// TwinCAT 3 PLC project FMS_201_Monol_tico
// ProgramVersion: 3.1.4024.0
// libraries:
//   Tc2_Standard, * (Beckhoff Automation GmbH)
//   Tc2_System, * (Beckhoff Automation GmbH)
//   Tc3_Module, * (Beckhoff Automation GmbH)
// project tree:
//   / PlcTask.TcTTO
//   POUs/ FB_Clock.TcPOU, FB_Estacion.TcPOU, MAIN.TcPOU (not stored)
// (motion and I/O tree: see PLC project fms_201_manual)
// real-time tasks:
//   TASK PlcTask: cycle T#10ms, priority 20, ADS port 350
//   TASK PlcTask1: cycle T#10ms, priority 21, ADS port 351
//   TASK PlcTask2: cycle T#10ms, priority 22, ADS port 352
//   TASK PlcTask3: cycle T#10ms, priority 23, ADS port 353
//   TASK PlcTask4: cycle T#10ms, priority 24, ADS port 354
//   TASK PlcTask5: cycle T#10ms, priority 25, ADS port 355
//   TASK PlcTask6: cycle T#10ms, priority 26, ADS port 356
// variable links:

CONFIGURATION FMS_201_Monol_tico
    RESOURCE PLC ON TwinCAT3
        TASK PlcTask(INTERVAL := T#10ms, PRIORITY := 23);
        PROGRAM MAIN WITH PlcTask : MAIN;
    END_RESOURCE
END_CONFIGURATION

// ---- POUs/FB_Clock.TcPOU
FUNCTION_BLOCK FB_Clock

VAR_INPUT
	EN: BOOL :=TRUE; 		// Entrada de nuestro temporizador
	PT: TIME := T#500MS;	// Tiempo de nuestro temporizador
END_VAR

VAR_OUTPUT
	ET: TIME;	// Sirve para consultar el tiempo que lleva la entrada PT
	Q: BOOL;	// Salida de nuestro temporizador
END_VAR
VAR
	Timer: TON;
END_VAR

// Función de salida

IF Timer.Q THEN
	Q := NOT Q;
END_IF

// Bloque de función TON
// Definimos la condición de entrada IN cuando EN esté TRUE (siempre) y no esté activa la salida del temporizador
Timer(IN:= EN AND NOT Timer.Q, PT := PT, ET => ET);

END_FUNCTION_BLOCK

// ---- POUs/FB_Estacion.TcPOU
FUNCTION_BLOCK FB_Estacion
VAR_INPUT
	// Parámetros
	TpoEstabilidad: TIME := T#2000MS;
	UdsSolicitadas:UINT := 5;
	
END_VAR
VAR_OUTPUT
	// Parámetros
	CondicionInicial: BOOL;
	UdsPendientes: UINT;
	UdsRealizadas: UINT;
	
	// Entradas comunes
	PulsadorEmergencia AT %I*: BOOL;
    SelectorManual AT %I*: BOOL;
    PulsadorMarcha AT %I*: BOOL;
    PulsadorParada AT %I*: BOOL := TRUE; // Contacto normalmente cerrado
    EstacionConectada AT %I*: BOOL := TRUE;
    DetectorPresion AT %I*: BOOL := TRUE;
	
	PalePresencia AT %I*: BOOL;
    PaleCodigoBit0 AT %I*: BOOL;
    PaleCodigoBit1 AT %I*: BOOL;
    PaleCodigoBit2 AT %I*: BOOL;
	
	// Entradas específicas
	DescargadorDetras AT %I*: BOOL;
	DescargadorDelante AT %I*: BOOL;
	VerticalArriba AT %I*: BOOL;
	VerticalAbajo AT %I*: BOOL;
	VerificadorArriba AT %I*: BOOL;
	VerificadorAbajo AT %I*: BOOL;
	DesplazadorDetras AT %I*: BOOL;
	AlimentadorDetras AT %I*: BOOL;
	AlimentadorDelante AT %I*: BOOL;
	VacioDescargador AT %I*: BOOL;
	PresenciaBaseAlimentador AT %I*:BOOL;
END_VAR
VAR
	// Bloques funcionales
	CLK: FB_Clock;
	// Salidas comunes
	DesconectaEstacion AT %Q*: BOOL;
    LamparaAlarma AT %Q*: BOOL;
    LamparaMarcha AT %Q*: BOOL;
	LamparaFaltaMaterial AT %Q*: BOOL;
    AvisadorSonoro AT %Q*: BOOL;

    CintaMotorActiva AT %Q*: BOOL;
    CintaMotorInvierte AT %Q*: BOOL;
    CintaRetenedorBaja AT %Q*: BOOL;
    CintaSeparadorSube AT %Q*: BOOL;
	
	// Salidas específicas
	DescargadorAtras AT %Q*: BOOL;
	DescargadorAdelante AT %Q*: BOOL;
	DescargadorBaja AT %Q*: BOOL;
	RechazadorAdelante AT %Q*: BOOL;
	VerificadorBaja AT %Q*: BOOL;
	DesplazadorAdelante AT %Q*: BOOL;
	AlimentadorAdelante AT %Q*: BOOL;
	EyectorSucciona AT %Q*: BOOL;
END_VAR

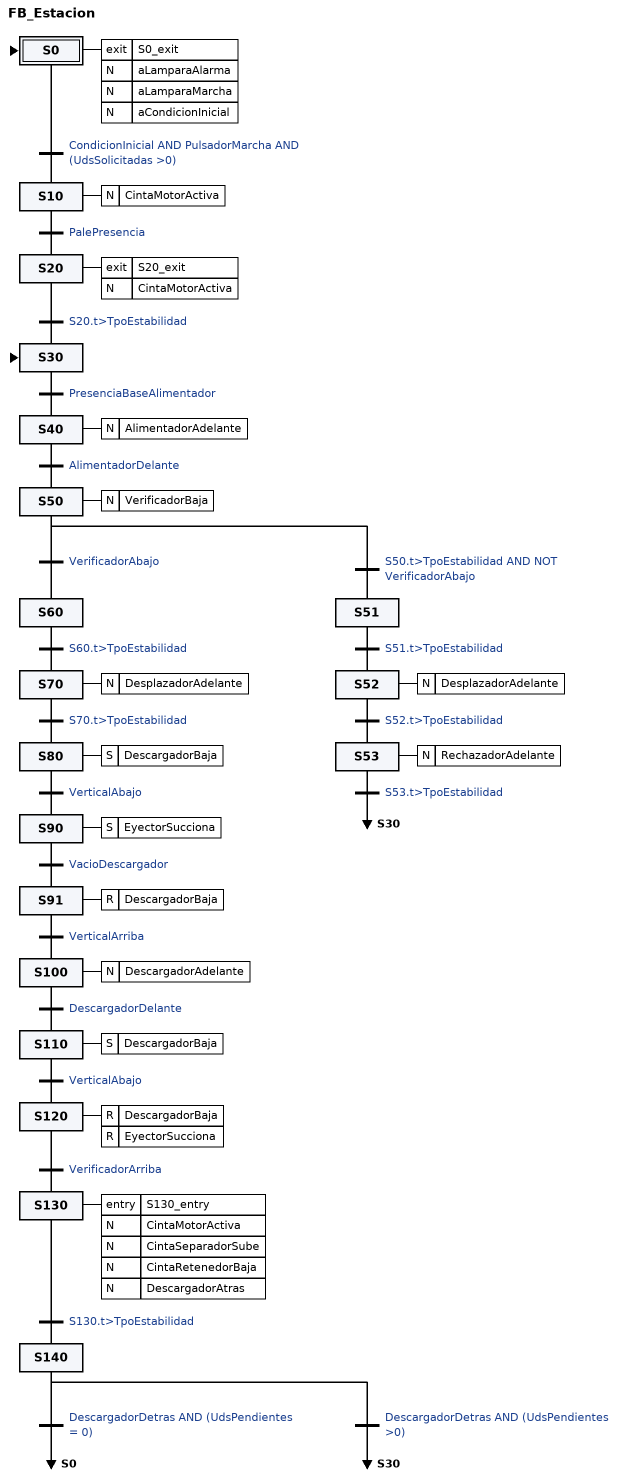
INITIAL_STEP S0:
    S0_exit(P0);  // exit action
    aLamparaAlarma(N);
    aLamparaMarcha(N);
    aCondicionInicial(N);
END_STEP
TRANSITION FROM S0 TO S10
    := CondicionInicial AND PulsadorMarcha AND (UdsSolicitadas >0);
END_TRANSITION
STEP S10:
    CintaMotorActiva(N);
END_STEP
TRANSITION FROM S10 TO S20
    := PalePresencia;
END_TRANSITION
STEP S20:
    S20_exit(P0);  // exit action
    CintaMotorActiva(N);
END_STEP
TRANSITION FROM S20 TO S30
    := S20.t>TpoEstabilidad;
END_TRANSITION
STEP S30:
END_STEP
TRANSITION FROM S30 TO S40
    := PresenciaBaseAlimentador;
END_TRANSITION
STEP S40:
    AlimentadorAdelante(N);
END_STEP
TRANSITION FROM S40 TO S50
    := AlimentadorDelante;
END_TRANSITION
STEP S50:
    VerificadorBaja(N);
END_STEP
TRANSITION FROM S50 TO S60
    := VerificadorAbajo;
END_TRANSITION
TRANSITION FROM S50 TO S51
    := S50.t>TpoEstabilidad AND NOT VerificadorAbajo;
END_TRANSITION
STEP S51:
END_STEP
TRANSITION FROM S51 TO S52
    := S51.t>TpoEstabilidad;
END_TRANSITION
STEP S52:
    DesplazadorAdelante(N);
END_STEP
TRANSITION FROM S52 TO S53
    := S52.t>TpoEstabilidad;
END_TRANSITION
STEP S53:
    RechazadorAdelante(N);
END_STEP
TRANSITION FROM S53 TO S30
    := S53.t>TpoEstabilidad;
END_TRANSITION
STEP S60:
END_STEP
TRANSITION FROM S60 TO S70
    := S60.t>TpoEstabilidad;
END_TRANSITION
STEP S70:
    DesplazadorAdelante(N);
END_STEP
TRANSITION FROM S70 TO S80
    := S70.t>TpoEstabilidad;
END_TRANSITION
STEP S80:
    DescargadorBaja(S);
END_STEP
TRANSITION FROM S80 TO S90
    := VerticalAbajo;
END_TRANSITION
STEP S90:
    EyectorSucciona(S);
END_STEP
TRANSITION FROM S90 TO S91
    := VacioDescargador;
END_TRANSITION
STEP S91:
    DescargadorBaja(R);
END_STEP
TRANSITION FROM S91 TO S100
    := VerticalArriba;
END_TRANSITION
STEP S100:
    DescargadorAdelante(N);
END_STEP
TRANSITION FROM S100 TO S110
    := DescargadorDelante;
END_TRANSITION
STEP S110:
    DescargadorBaja(S);
END_STEP
TRANSITION FROM S110 TO S120
    := VerticalAbajo;
END_TRANSITION
STEP S120:
    DescargadorBaja(R);
    EyectorSucciona(R);
END_STEP
TRANSITION FROM S120 TO S130
    := VerificadorArriba;
END_TRANSITION
STEP S130:
    S130_entry(P1);  // entry action
    CintaMotorActiva(N);
    CintaSeparadorSube(N);
    CintaRetenedorBaja(N);
    DescargadorAtras(N);
END_STEP
TRANSITION FROM S130 TO S140
    := S130.t>TpoEstabilidad;
END_TRANSITION
STEP S140:
END_STEP
TRANSITION FROM S140 TO S0
    := DescargadorDetras AND (UdsPendientes = 0);
END_TRANSITION
TRANSITION FROM S140 TO S30
    := DescargadorDetras AND (UdsPendientes >0);
END_TRANSITION

ACTION aCondicionInicial:
CondicionInicial:= EstacionConectada AND AlimentadorDetras AND DesplazadorDetras  AND VerificadorArriba AND DescargadorDetras;
END_ACTION

ACTION aLamparaAlarma:
LamparaAlarma := (S0.x AND NOT CondicionInicial AND CLK.Q);
END_ACTION

ACTION aLamparaMarcha:
LamparaMarcha := (S0.x AND CondicionInicial AND CLK.Q) OR NOT S0.x;

CLK();
END_ACTION

ACTION S0_exit:
// Actualizamos el número de uds cada vez que se inicia
IF (UdsPendientes = 0) THEN
	UdsPendientes := UdsSolicitadas;
END_IF
END_ACTION

ACTION S130_entry:
// Al completar correctamente la transferencia
// Actualizamos el número de unidades realizadas
UdsRealizadas := UdsRealizadas + 1;

// Si quedan unidades pendientes actualizamos también su valor
IF (UdsPendientes >0) THEN
	UdsPendientes := UdsPendientes -1;
END_IF
END_ACTION

ACTION S20_exit:

END_ACTION

END_FUNCTION_BLOCK
